// TIA Portal V20 export
FUNCTION_BLOCK "Conveyor_C1"   // FB2, LAD
TITLE = New Title
// stored: Access Published, MemoryReserve 100, SetENOAutomatically false
   VAR
      jogRight : Bool;
   END_VAR
BEGIN

REGION Network 1: Run conveyor LEFT
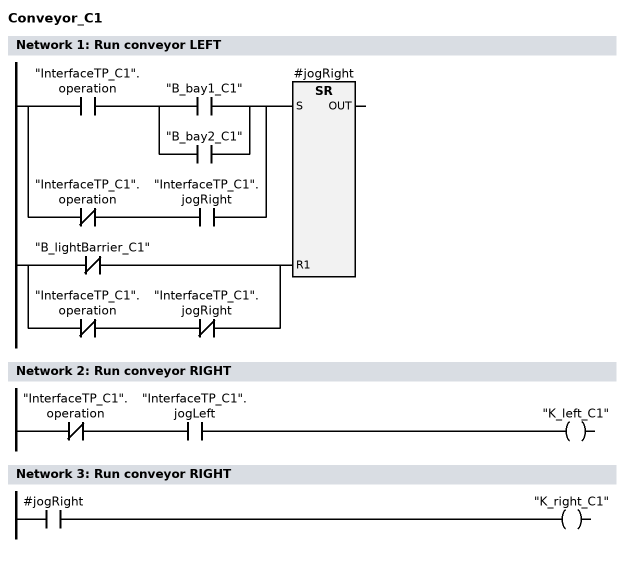
   RUNG wire#powerrail
      Contact( "InterfaceTP_C1".operation )
      wire#w1
      Contact( "B_bay1_C1" )
      wire#w2
      S_SR(operand := #jogRight, r1 := wire#w3)
   END_RUNG
   RUNG wire#w1
      Contact( "B_bay2_C1" )
   END_RUNG wire#w2
   RUNG wire#powerrail
      I_Contact( "InterfaceTP_C1".operation )
      Contact( "InterfaceTP_C1".jogRight )
   END_RUNG wire#w2
   RUNG wire#powerrail
      I_Contact( "B_lightBarrier_C1" )
   END_RUNG wire#w3
   RUNG wire#powerrail
      I_Contact( "InterfaceTP_C1".operation )
      I_Contact( "InterfaceTP_C1".jogRight )
   END_RUNG wire#w3
   // the same network as SCL:
   IF ("InterfaceTP_C1".operation AND ("B_bay1_C1" OR "B_bay2_C1")) OR (NOT "InterfaceTP_C1".operation AND "InterfaceTP_C1".jogRight) THEN
       #jogRight := TRUE;   // SR flip-flop
   END_IF;
   IF NOT "B_lightBarrier_C1" OR (NOT "InterfaceTP_C1".operation AND NOT "InterfaceTP_C1".jogRight) THEN
       #jogRight := FALSE;
   END_IF;
END_REGION

REGION Network 2: Run conveyor RIGHT
   RUNG wire#powerrail
      I_Contact( "InterfaceTP_C1".operation )
      Contact( "InterfaceTP_C1".jogLeft )
      Coil( "K_left_C1" )
   END_RUNG
   // the same network as SCL:
   "K_left_C1" := NOT "InterfaceTP_C1".operation AND "InterfaceTP_C1".jogLeft;
END_REGION

REGION Network 3: Run conveyor RIGHT
   RUNG wire#powerrail
      Contact( #jogRight )
      Coil( "K_right_C1" )
   END_RUNG
   // the same network as SCL:
   "K_right_C1" := #jogRight;
END_REGION
END_FUNCTION_BLOCK
